TYPE ParIDAccess_Status_typ : 	
	STRUCT 
		Done : BOOL;
		Busy : BOOL;
		CommandAborted : BOOL;
		Active : BOOL ;
	END_STRUCT
END_TYPE

(* stored: Version 1.1.0.1, ProductVersion 3.1.4024.3
   DUT ParIDAccess_Status_typ: Id {08c11d28-c3ba-028a-14bc-bf87ee88b168} *)
